{attribute 'qualified_only'}
{attribute 'strict'}
{attribute 'to_string'}
TYPE E_EventType :
(
	Information		:= 1,
	Warning			:= 2,
	Stop			:= 3,
	Abort			:= 4
);
END_TYPE

(* stored: Version 1.1.0.1
   DUT E_EventType: Id {8295607b-d518-0b57-3eba-11dbcbeb4051} *)
